Staubli VAL3: recursion2.pgx

program recursion2(string& x_sString (dimensions=1))
begin
  nNum=nNum+1
  call recursion2(sString)

end
